FUNCTION_BLOCK FB_R_TRIG (* Detect rising edge *)
  PACKAGE iec61131::edgeDetection;
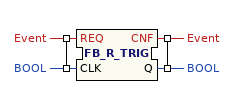
  EVENT_INPUT
    REQ WITH CLK; (* Normal Execution Request *)
  END_EVENT
  EVENT_OUTPUT
    CNF WITH Q; (* Execution Confirmation *)
  END_EVENT
  VAR_INPUT
    CLK : BOOL; (* Clock *)
  END_VAR
  VAR_OUTPUT
    Q : BOOL; (* Output *)
  END_VAR
  VAR
    MEM : BOOL;
  END_VAR
  ALGORITHM REQ IN ST:
Q := CLK AND NOT MEM;
MEM := CLK;
  END_ALGORITHM
END_FUNCTION_BLOCK
